INTERFACE I_JsonLanguagePack

METHOD PUBLIC AddDataTypeConversionUsingConverter
VAR_INPUT
	DataType : T_MAXSTRING;
	TypeConversion : I_JsonTypeConverter;
END_VAR
END_METHOD

METHOD PUBLIC AddDataTypeConversionUsingVariable
VAR_INPUT
	DataType : T_MAXSTRING;
	VariableOfType : ANY;
END_VAR
END_METHOD

METHOD PUBLIC DataToJsonString : HRESULT
VAR_INPUT
	Source : I_DataAccess;
	JsonStringAddress : POINTER TO STRING;
	JsonStringSize : UDINT;
END_VAR
END_METHOD

METHOD PUBLIC DataToJsonStringSize : UDINT
VAR_INPUT
	Source : I_DataAccess;
END_VAR
END_METHOD

METHOD PUBLIC Install
VAR_INPUT
	DataTypePack : I_JsonDataTypePack;
END_VAR
END_METHOD

METHOD PUBLIC JsonStringToData : I_DataDisposer
VAR_INPUT
	JsonStringPointer : POINTER TO STRING;
	Destination : I_DataAccess;
END_VAR
END_METHOD

END_INTERFACE

(* stored: Version 1.1.0.1, ProductVersion 3.1.4024.12
   Itf I_JsonLanguagePack: Id {d16ff96f-90eb-09d8-1b98-c2706e79cd45}
   Method AddDataTypeConversionUsingConverter: Id {f361b5d7-b6f0-02ab-04e6-e6a1298f8013}
   Method AddDataTypeConversionUsingVariable: Id {d11a36c3-04c8-086b-020a-9306fdc45644}
   Method DataToJsonString: Id {74afc927-4797-0027-0ca7-b1ef216f101b}
   Method DataToJsonStringSize: Id {05055305-1f06-071c-26d1-d0ae6576dada}
   Method Install: Id {47911e50-4ffd-0129-0736-e738ee235dff}
   Method JsonStringToData: Id {072d9472-c573-0613-1c2c-08870beeb6de} *)
